PROGRAM MAIN
VAR

	bVISSafetyResetIn: BOOL;
END_VAR

(*
bSafetyReset:=bSafetyResetIn OR bVISSafetyResetIn;
bErrorAck:=bSafetyResetIn OR bVISSafetyResetIn;
bSafetyReset2:=bSafetyResetIn OR bVISSafetyResetIn;

*)
P_SAFETY();

//Sygnały dla ProgramPLC
QbEmergencyStopButton:=bEmergencyStopButton;
QbEmergencyStop:=bEmergencyStop;
QbBottleFeederSafety:=bBottleFeederSafety;
//Na potrzeby rygli
bSafetyResetOut :=	bSafetyResetIn OR bPucksInserterSafetyResetIn OR bSafetyResetInRC40;

END_PROGRAM

(* stored: Version 1.1.0.1, ProductVersion 3.1.4026.13, FileIdentifier 9820b9c5917a6ae1bc75e6323b0ca7e1feee96f0, FileSignature 3c1259b87e9c697f5bd9cf36df24746f4fc4d851898abf19f82e60f18ac4d122e16e19f1f564b1292fbbac7f365c34144470df2867655ef238e28ece2d4bb3eab31ce817ac95b340b787d0d77b0e74942eb0d72e2bdef4cf1457bfff68bfc1c8c6e746577ce9e679ed7207fbc5184929bb5439a3d752fe236a67051a057fbe9988a63cef7577168dfc106a6dd1007cec65544aba33c22681332a271fc0bed784662cb202f7d8076543f77f369eda30028324f4a8cc4a58712783acf46f316554676e3936103829313b8e795d7a07a3dd22e2739eb74bf96ea6a74899901187029b3c6e2d04145e3156401bf1538776e6003dcbd750d45586a6a9f9d8e39e674d
   POU MAIN: Id {85b14d12-419a-4ef1-bed1-c0aa7ef3e2a3}, SpecialFunc None *)
